// TIA Portal V17 export
// export: Created 2025-03-07T09:17:01.2285428Z, ExportSetting WithDefaults, DisplayName Totally Integrated Automation Portal, DisplayVersion V17 Update 8, DisplayName TIA Portal Openness, DisplayVersion V17 Update 8, DisplayName TIA Portal Version Control Interface, DisplayVersion V17, DisplayName SINAMICS Startdrive Advanced, DisplayVersion V17 SP2, DisplayName SINAMICS Startdrive G110M, G120, G120C, G120D, G120P, G115D, DisplayVersion V17 SP2, DisplayName SINAMICS Startdrive G130, G150, S120, S150, SINAMICS MV, S210, DisplayVersion V17 SP2, DisplayName STEP 7 Professional, DisplayVersion V17 Update 8, DisplayName SINUMERIK ONE STEP 7 Toolbox, DisplayVersion V17 Update 12, DisplayName SINUMERIK 840D sl STEP 7 Toolbox, DisplayVersion V17 Update 12, DisplayName STEP 7 Safety, DisplayVersion V17 Update 6, DisplayName WinCC Advanced, DisplayVersion V17 Update 8
DATA_BLOCK "DB7339_ROBOT_CELL_TEST_INTERLOCK"   // DB7339
{ S7_Optimized_Access := 'FALSE'; DB_Accessible_From_OPC_UA := 'FALSE' }
AUTHOR : ETXETAR
VERSION : 1.0
// stored: AutoNumber false, DBAccessibleFromOPCUA false, DBAccessibleFromWebserver true, IsOnlyStoredInLoadMemory false, IsWriteProtectedInAS false
   VAR RETAIN
      INTERLOCKS : Struct
         OUT_OF_INTERFERENCE : Bool;   // OUT OF INTERFERANCE
         ENABLE_OPEN_SAFE_DR_MC : Bool := true;   // ENABLE OPEN SAFETY MACHINE DOOR
         RUN_OUT_REQUESTED : Bool;   // RUNOUT REQUESTED
         PART_TYPE_CHANGE_OVER : Bool;   // PART TYPE CHANGE OVER
         STOP_END_OF_CYCLE : Bool;   // STOP END OF CYCLE (GANTRY TEST) / STOP END OF CYCLE
         EMERGENCY_STOP : Bool := true;   // EMERGENCY STOP
         PART_ID_1 : Array[0..63] of Byte;   // PART ID 1
         PART_ID_2 : Array[0..63] of Byte;   // PART ID 2
         PART_ID_3 : Array[0..63] of Byte;   // PART ID 3
      END_STRUCT;
   END_VAR
BEGIN
END_DATA_BLOCK
